// TwinCAT 3 PLC project _00_Strategy
// ProgramVersion: 3.1.4023.0
// libraries:
//   Tc2_Standard, * (Beckhoff Automation GmbH)
//   Tc2_System, * (Beckhoff Automation GmbH)
//   Tc3_Module, * (Beckhoff Automation GmbH)
// project tree:
//   Helpers/ C_TO_F.TcPOU, RES_PT.TcPOU, TEMP_PT.TcPOU
//   / MAIN.TcPOU, PlcTask.TcTTO
//   Strategy Pattern/Motors/ motor.TcPOU
//   Strategy Pattern/ P_Strategy.TcPOU (not stored)
//   Strategy Pattern/Temperature sensor/ ITempSensor.TcIO (not stored), tempSensor.TcPOU, tempSensor_PT100.TcPOU, tempSensor_PT1000.TcPOU (not stored)
// (motion and I/O tree: see PLC project 13_decorator)
// real-time tasks:
//   TASK PlcTask: cycle T#10ms, priority 20, ADS port 350
// variable links:

CONFIGURATION _00_Strategy
    RESOURCE PLC ON TwinCAT3
        TASK PlcTask(INTERVAL := T#10ms, PRIORITY := 20);
        PROGRAM MAIN WITH PlcTask : MAIN;
    END_RESOURCE
END_CONFIGURATION

// ---- MAIN.TcPOU
PROGRAM MAIN
VAR
END_VAR

(* 
	GOF 		Define a family of algorithms, encapsulate each one, and make them interchangeable.
				Strategy lets the algorithm vary independently from clients using it.   
*)
P_Strategy();

END_PROGRAM

// ---- Helpers/C_TO_F.TcPOU
FUNCTION C_TO_F : REAL
VAR_INPUT
	celsius : REAL;
END_VAR


(*
version 1.1	11. mar. 2009
programmer 	hugo
tested by		tobias

this function converts celsius  to fahrenheit 

*)

C_TO_F := celsius * 1.8 + 32.0;


(* revision history

hm	4. aug. 2006	rev 1.0
	original version

hm	11. mar. 2009	rev 1.1
	real constants updated to new systax using dot

*)

END_FUNCTION

// ---- Helpers/RES_PT.TcPOU
FUNCTION RES_PT : REAL
VAR_INPUT
	T : REAL;
	R0 : REAL;
END_VAR
VAR CONSTANT
	A : REAL := 3.90802E-3 ;
	B : REAL := -5.802E-7;
	C : REAL := -4.27350E-12;
END_VAR
VAR
	T2: REAL;
END_VAR

(*
version 1.3	11. mar. 2009
programmer 	hugo
tested by		oscat


this function returs the resistance for a platinum sensor for a temperature range from -200..+850 °C *)

T2 := T * T;

IF T >= 0.0 THEN
	RES_PT := R0 * ( 1.0 + A * T + B * T2);
ELSE
	RES_PT := R0 * ( 1.0 + A * T + B * T2 + C * (T - 100.0) * T2 * T);
END_IF;



(* revision history
hm	4. aug. 2006	rev 1.1
	original version

hm	2. dec 2007	rev 1.2
	changed code for better performance

hm	11. mar. 2009	rev 1.3
	changed real constants to use dot syntax

*)


(*
 Auszug aus DIN 43760 für Pt100

°C		R		°C		R		°C	R			°C		R			°C		R			°C		R

-200 	18,49 	-100 	60,25 	0 	100,00 	100 	138,50 	200 	175,84 	300 	212,02
-195 	20,65 	-95 	62,28 	5 	101,95 	105 	140,39 	205 	177,68 	305 	213,80
-190 	22,80 	-90 	64,30 	10 	103,90 	110 	142,29 	210 	179,51 	310 	215,57
-185 	24,94 	-85 	66,31 	15 	105,85 	115 	144,17 	215 	181,34 	315 	217,35
-180 	27,08 	-80 	68,33 	20 	107,79 	120 	146,06 	220 	183,17 	320 	219,12
-175 	29,20 	-75 	70,33 	25 	109,73 	125 	147,94 	225 	184,99 	325 	220,88
-170 	31,32 	-70 	72,33 	30 	111,67 	130 	149,82 	230 	186,82 	330 	222,65
-165 	33,43 	-65 	74,33 	35 	113,61 	135 	151,70 	235 	188,63 	335 	224,41
-160 	35,33 	-60 	76,33 	40 	115,54 	140 	153,58 	240 	190,45 	340 	226,17
-155 	37,63 	-55 	78,32 	45 	117,47 	145 	155,45 	245 	192,26 	345 	227,92
-150 	39,71 	-50 	80,31 	50 	119,40 	150 	157,31 	250 	194,07 	350 	229,67
-145 	41,79 	-45 	82,29 	55 	121,32 	155 	159,18 	255 	195,88 	355 	231,42
-140 	43,87 	-40 	84,27 	60 	123,24 	160 	161,04 	260 	197,69 	360 	233,17
-135 	45,94 	-35 	86,25 	65 	125,16 	165 	162,90 	265 	199,49 	365 	234,91
-130 	48,00 	-30 	88,22 	70 	127,07 	170 	164,76 	270 	201,29 	370 	236,65
-125 	50,06 	-25 	90,19 	75 	128,98 	175 	166,61 	275 	203,08 	375 	238,39
-120 	52,11 	-20 	92,16 	80 	130,89 	180 	168,46 	280 	204,88 	380 	240,13
-115 	54,15 	-15 	94,12 	85 	132,80 	185 	170,31 	285 	206,67 	385 	241,86
-110 	56,19 	-10 	96,09 	90 	134,70 	190 	172,16 	290 	208,45 	390 	243,59
-105 	58,22 	-5 		98,04 	95 	136,60 	195 	174,00 	295 	210,24 	395 	245,31

*)
(*
revision history


*)

END_FUNCTION

// ---- Helpers/TEMP_PT.TcPOU
FUNCTION TEMP_PT : REAL
VAR_INPUT
	Res : REAL;
	R0 : REAL;
END_VAR
VAR CONSTANT
	A : REAL := 3.9083E-3 ;
	B : REAL := -5.775E-7;
	accuracy : REAL := 0.01;
END_VAR
VAR
	step: REAL := 50.0;
	X: REAL;
	Y: REAL;
	t1: REAL;
	pt : POINTER TO DWORD;
END_VAR
(*
version 1.7	11. mar. 2009
programmer 	hugo
tested by		oscat

this function returs the temperature for a platinum sensor for a range from -200..+850 °C *)

X := A * R0;
Y := B * R0;
IF Res >= R0 THEN
	t1 := X * X - 4.0 * Y * (R0 - Res);
	IF t1 < 0.0 THEN
		TEMP_PT := 10000.0;
	ELSE
		TEMP_PT := (-X + SQRT(t1)) / (2.0 * Y);
	END_IF;
ELSE
	pt := ADR(step);
	(* since the formula cannot be solved this is a successive approximation *)
	TEMP_PT := -100.0;
	WHILE step > accuracy DO
		(* test if result greater or less *)
		IF RES_PT(TEMP_PT, R0) < res THEN TEMP_PT := TEMP_PT + step; ELSE TEMP_PT := TEMP_PT - step; END_IF;
		pt^ := pt^ - 8388608;  (* this is a super fast divide by 2 method for non floating point CPUs *)
		(* the alternative code: step := step * 0.5; *)
	END_WHILE;
END_IF;

(* revision history

rev 1.1 hm 24.1.2007	
	deleted unused variable C

rev 1.2 hm 10.9.2007
	reduced accuracy to 0.02 to shorten execution time

rev 1.3	hm	2. dec 2007
	changed code for better performance

rev	1.4	hm	23. dec 2007
	avoid a negative square root if input values are wrong

rev 1.5 hm	5. jan 2008
	replaced / 2 with * 0.5 for better performance

hm	31. oct. 2008	rev 1.6
	improved performance

hm	11. mar. 2009	rev 1.7
	changed real constants to use dot syntax

*)

END_FUNCTION

// ---- Strategy Pattern/Motors/motor.TcPOU
{attribute 'no_explicit_call' := 'This is a CLASS and should be accessed using methods or properties'}
FUNCTION_BLOCK motor
VAR
	// The concrete temperature sensor interface pointer is set
	// 	* during FB_Init
	//  * during runtime via property changeTempSensor  
	_tempSensor					: ITempSensor;
END_VAR

(*  
	Principally a CLASS should be accessed using methods or properties
	Good practice is not put code here, or call the class directly 
	Or maybe just a call to a method calling the cyclic code 
*)
cyclicCall();

// Change the concrete temperature sensor interface pointer during runtime  
PROPERTY changeTempSensor : ITempSensor
SET
// Change the concrete temperature sensor interface pointer during runtime  
_tempSensor := changeTempSensor;
END_SET
END_PROPERTY

METHOD cyclicCall
;
END_METHOD

METHOD FB_Init : BOOL
VAR_INPUT
    bInitRetains 			: BOOL ; // if TRUE, the retain variables are initialized (reset warm / reset cold)
    bInCopyCode  			: BOOL ; // if TRUE, the instance afterwards gets moved into the copy code (online change)
	tempSensor				: ITempSensor;
END_VAR
// Set the concrete temperature sensor interface pointer during instantiation of the class  
this^._tempSensor := tempSensor;
END_METHOD

PROPERTY motorTemperature : real
GET
// Our implementation requires temperature feedback in degrees Celcius
motorTemperature := _tempSensor.tempDegreesC;
END_GET
END_PROPERTY

END_FUNCTION_BLOCK

// ---- Strategy Pattern/Temperature sensor/tempSensor.TcPOU
{attribute 'no_explicit_call' := 'This is a CLASS and should be accessed using methods or properties'}
FUNCTION_BLOCK tempSensor IMPLEMENTS ITempSensor
VAR
	rawValue			AT %I*	: INT;		// measurement value of sensor
END_VAR
(*~
<docu>
	<summary>
			Implementation of a Temperature sensor class
			
			The base class returns the raw value / 10
			
			Usage as follows :
			<code>
				FUNCTION_BLOCK concreteTempSensor
			</code>
	</summary>				
</docu>	
~*)

(*  
	Principally a CLASS should be accessed using methods or properties
	Good practice is not put code here, or call the class directly 
	Or maybe just a call to a method calling the cyclic code 
*)

PROPERTY DEBUG_setRawValue : int
SET
rawValue := DEBUG_setRawValue;
END_SET
END_PROPERTY

PROPERTY tempDegreesC : REAL
GET
// Returns the value of the terminal / 10
tempDegreesC := TO_REAL(rawValue) / 10.0;
END_GET
END_PROPERTY

PROPERTY tempDegreesF : REAL
GET
tempDegreesF := C_TO_F(celsius:=tempDegreesC);
END_GET
END_PROPERTY

END_FUNCTION_BLOCK

// ---- Strategy Pattern/Temperature sensor/tempSensor_PT100.TcPOU
{attribute 'no_explicit_call' := 'This is a CLASS and should be accessed using methods or properties'}
FUNCTION_BLOCK tempSensor_PT100 EXTENDS tempSensor
(*~
<docu>
	<summary>
			Implementation of a PT100 Temperature sensor class based on the base class tempSensor

			Usage:
			degreesC / degreesF return the Celcius / Fahrenheit value determined by the appropriate formula 		
	</summary>				
</docu>	
~*)

(*  
	Principally a CLASS should be accessed using methods or properties
	Good practice is not put code here, or call the class directly 
	Or maybe just a call to a method calling the cyclic code 
*)

PROPERTY tempDegreesC : REAL
GET
tempDegreesC := TEMP_PT(
			Res	:= TO_REAL(rawValue), 
			R0	:= 100.0
			);
END_GET
END_PROPERTY

END_FUNCTION_BLOCK
